TYPE TcoCylinderStatus :
STRUCT
	ActionDescription : STRING(100);	
END_STRUCT
END_TYPE

(* stored: Version 1.1.0.1
   DUT TcoCylinderStatus: Id {9207b296-4774-41cf-81ec-9938e823891e} *)
